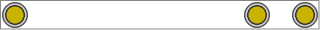
VISUALIZATION CtrlAxisInput  // 320x30
VAR_INPUT
	In:							UDINT;
END_VAR
    Lamp1 (0,0 30x30), variable: In.0, style: Lamp-Lamp1-Yellow
    Lamp1 (242,0 30x30), variable: In.2, style: Lamp-Lamp1-Yellow
    Lamp1 (290,0 30x30), variable: In.1, style: Lamp-Lamp1-Yellow
END_VISUALIZATION

(* stored: Version 1.1.0.1, ProductVersion 3.1.4024.3
   Visu CtrlAxisInput: Id {6aecc89e-4e9f-4a48-bc1e-f87b2ea590d3} *)
